Fanuc KAREL source: ka00010.KL

-- PROVISIONAL review KL for V1013-1; original PC SHA256 0fcd886526b324bc8bc78801bec7b645f1febe39c8db6c34e96b29fc8dcefb56
-- Incomplete behavior may be omitted. Consult companion uncertainty JSON. Do not deploy.
PROGRAM KA00010
%NOLOCKGROUP
VAR
  SRC : INTEGER
-- UNRESOLVED_DECL DST type=00001c
BEGIN
  -- UNRESOLVED_PC offsets 5-16; opcodes 2E,23
  -- UNRESOLVED_PC offsets 21-33; opcodes 21,23
  -- UNRESOLVED_PC offsets 38-42; opcodes 7F
END KA00010
